FUNCTION CheckRangeInt : INT
VAR_INPUT
    InValue : INT;
END_VAR
VAR
END_VAR

IF InValue < 0 THEN
    CheckRangeInt := 0;
ELSIF InValue > 32767 THEN
    CheckRangeInt := 32767;
ELSE
    CheckRangeInt := InValue;
END_IF

END_FUNCTION

(* stored: Version 1.1.0.1, ProductVersion 3.1.4024.15
   POU CheckRangeInt: Id {a64d7b82-66be-44d2-a85d-c7c89efbe026}, SpecialFunc None *)
